(*
Function indside folder `ExampleFolder`.
*)
FUNCTION F_ExampleFolder_Function : BOOL

END_FUNCTION

(* stored: Version 1.1.0.1, ProductVersion 3.1.4024.11
   POU F_ExampleFolder_Function: Id {a8054540-25f8-4f51-9203-ddc488e3ec02}, SpecialFunc None *)
